# EPICS substitutions: db/Beckhoff_9XXX/ecmcEL9221-5000.substitutions
file "ecmcEL9221-5000-chX.template"
{
    pattern {CH_ID}
            {01   }
}
